// TwinCAT 3 PLC project PLC1
// ProgramVersion: 3.1.4024.0
// libraries:
//   Tc2_Standard, * (Beckhoff Automation GmbH)
//   Tc2_System, * (Beckhoff Automation GmbH)
//   Tc3_Module, * (Beckhoff Automation GmbH)
// project tree:
//   / PlcTask.TcTTO
//   POUs/ MAIN.TcPOU
// real-time tasks:
//   TASK PlcTask: cycle T#10ms, priority 20, ADS port 350
//   TASK Device 1 (OPC UA Virtual)_Task_58: cycle T#40ms, priority 58, ADS port 351
// I/O:
//   DEVICE Device 1 (OPC UA Virtual), AmsNetId 10.33.70.115.2.1
// variable links:
//   PLC1/PLC1 Instance <-> Device 1 (OPC UA Virtual)/Client #1
//     PlcTask Outputs/MAIN.opcua_client_write_enable <-> Outputs/Control/Write Enable
//   PLC1/PLC1 Instance <-> Device 1 (OPC UA Virtual)/Client #1/PLC1.MAIN.opcua_server_read
//     PlcTask Outputs/MAIN.opcua_client_write <-> Outputs/Value
//   PLC1/PLC1 Instance <-> Device 1 (OPC UA Virtual)/Client #1/PLC1.MAIN.opcua_server_write
//     PlcTask Inputs/MAIN.opcua_client_read <-> Inputs/Value

CONFIGURATION PLC1
    RESOURCE PLC ON TwinCAT3
        TASK PlcTask(INTERVAL := T#10ms, PRIORITY := 20);
        PROGRAM MAIN WITH PlcTask : MAIN;
    END_RESOURCE
END_CONFIGURATION

// ---- POUs/MAIN.TcPOU
PROGRAM MAIN
VAR
	{attribute 'OPC.UA.DA' := '1'}
	opcua_server_read 		: REAL;
	{attribute 'OPC.UA.DA' := '1'}
	opcua_server_write		: REAL;
	
	opcua_client_read				AT %I*	: REAL;
	opcua_client_write				AT %Q*	: REAL;
	opcua_client_write_enable 		AT %Q* : BOOL := TRUE;
	
END_VAR

END_PROGRAM
